ABB RobotStudio station: sesion2_parte1.rspag

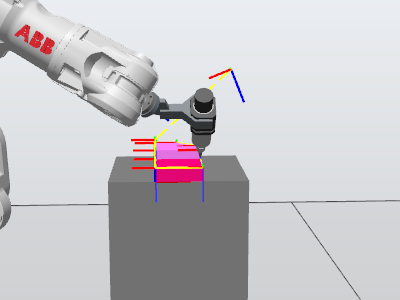
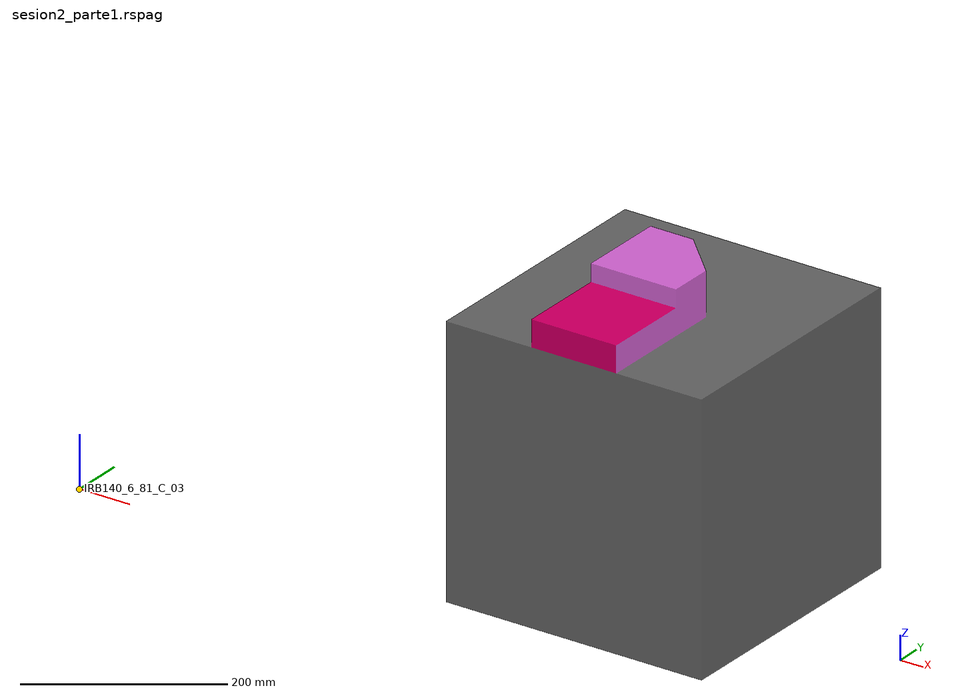
[picture v1: parts stored in the station drawn from their meshes, with robot base, taught points and paths (robot models come from the ABB library and are not in the file)]
--- station ---
Station sesion2 (saved by RobotStudio 24.1.10713.1)
Controller Controlador2
  mechanical unit ROB_1: IRB140_6_81_C_03, 6 joints, base frame (0, 0, 0) mm
Layout (positions relative to the parent item):
  - IRB140_6_81_C_03 [mechanism, from %ABB.RobotStudio.Models.IRB140%\IRB140_6_81_C_G_03.rslib] at (0, 0, 0) mm; joint values [-0.1632, 0.2338, 0.3026, 1.2516, 0.7538, -0.7373] (rad or m)
  - MyTool [mechanism, from Training Objects\myTool.rslib] at (513.67, -41.8, 471.8) mm, rotated rx 128.24 ry 25.81 rz 151.08 deg
  - Pieza_1 [part], size 300 x 300 x 300 mm
  - Pieza_7 [part], size 100 x 200 x 50 mm
Attachment: MyTool is attached to IRB140_6_81_C_03 / Link6
Attachment: Workobject_1 is attached to Pieza_7
Targets, tools, work objects and paths stored in the station and not in the controller backup, written as RAPID:
! task T_ROB1
MODULE CalibData
  PERS tooldata MyTool:=[TRUE,[[31.792631019,0,229.638935148],[0.945518576,0,0.325568154,0]],[1,[0,0,1],[1,0,0,0],0,0,0]];
  TASK PERS wobjdata Workobject_1:=[FALSE,TRUE,"",[[530,0,300],[1,0,0,0]],[[0,0,0],[1,0,0,0]]];
ENDMODULE

! task T_ROB1
MODULE Module1
  CONST robtarget Target_10:=[[0,0,30],[0,0,1,0],[0,0,-1,0],[9E+09,9E+09,9E+09,9E+09,9E+09,9E+09]];
  CONST robtarget Target_20:=[[100,0,30],[0,0,1,0],[0,0,-1,0],[9E+09,9E+09,9E+09,9E+09,9E+09,9E+09]];
  CONST robtarget Target_30:=[[100,100,30],[0,0,1,0],[0,-1,0,0],[9E+09,9E+09,9E+09,9E+09,9E+09,9E+09]];
  CONST robtarget Target_40:=[[100,100,50],[0,0,1,0],[0,-1,0,0],[9E+09,9E+09,9E+09,9E+09,9E+09,9E+09]];
  CONST robtarget Target_50:=[[100,150,50],[0,0,1,0],[0,-1,0,0],[9E+09,9E+09,9E+09,9E+09,9E+09,9E+09]];
  CONST robtarget Target_60:=[[50,200,50],[0,0,1,0],[0,-1,0,0],[9E+09,9E+09,9E+09,9E+09,9E+09,9E+09]];
  CONST robtarget Target_70:=[[0,200,50],[0,0,1,0],[0,-1,0,0],[9E+09,9E+09,9E+09,9E+09,9E+09,9E+09]];
  CONST robtarget Target_80:=[[0,100,50],[0,0,1,0],[0,-1,0,0],[9E+09,9E+09,9E+09,9E+09,9E+09,9E+09]];
  CONST robtarget Target_90:=[[0,100,30],[0,0,1,0],[0,-1,0,0],[9E+09,9E+09,9E+09,9E+09,9E+09,9E+09]];
  CONST robtarget pAprox:=[[0,0,90],[0,0,1,0],[0,0,-1,0],[9E+09,9E+09,9E+09,9E+09,9E+09,9E+09]];
  CONST robtarget pReposo:=[[689.268566117,0,537.147256028],[0.190808934,0,0.981627195,0],[0,0,0,0],[9E+09,9E+09,9E+09,9E+09,9E+09,9E+09]];
  CONST robtarget Target_30_Girado:=[[100,100,30],[0,0,0.923879533,0.382683432],[-1,0,-1,0],[9E+09,9E+09,9E+09,9E+09,9E+09,9E+09]];
  CONST robtarget Target_40_girado:=[[100,100,50],[0,0,0.923879533,0.382683432],[-1,0,-1,0],[9E+09,9E+09,9E+09,9E+09,9E+09,9E+09]];
  PROC Path_10()
    MoveJ pReposo,v1500,z100,MyTool\WObj:=wobj0;
    MoveJ pAprox,v1000,z100,MyTool\WObj:=Workobject_1;
    MoveL Target_10,v50,z0,MyTool\WObj:=Workobject_1;
    MoveL Target_20,v50,z0,MyTool\WObj:=Workobject_1;
    MoveL Target_30,v50,z0,MyTool\WObj:=Workobject_1;
    MoveL Target_30_Girado,v10,z0,MyTool\WObj:=Workobject_1;
    MoveL Target_40_girado,v50,z0,MyTool\WObj:=Workobject_1;
    MoveL Target_40,v50,z0,MyTool\WObj:=Workobject_1;
    MoveL Target_50,v50,z0,MyTool\WObj:=Workobject_1;
    MoveL Target_60,v50,z0,MyTool\WObj:=Workobject_1;
    MoveL Target_70,v50,z0,MyTool\WObj:=Workobject_1;
    MoveL Target_80,v50,z0,MyTool\WObj:=Workobject_1;
    MoveL Target_90,v50,z0,MyTool\WObj:=Workobject_1;
    MoveL Target_10,v50,z0,MyTool\WObj:=Workobject_1;
    MoveL pAprox,v50,z0,MyTool\WObj:=Workobject_1;
    MoveJ pReposo,v1000,z100,MyTool\WObj:=wobj0;
  ENDPROC
ENDMODULE


--- Backups/Controlador2/RAPID/TASK1/PROGMOD/Module1.mod ---
MODULE Module1
    !***********************************************************
    !
    ! M?dulo:  Module1
    !
    ! Descripción:
    !   <Introduzca la descripción aquí>
    !
    ! Autor: yisus
    !
    ! Versión: 1.0
    !
    !***********************************************************


    !***********************************************************
    !
    ! Procedimiento Main
    !
    !   Este es el punto de entrada de su programa
    !
    !***********************************************************
    PROC main()
        !Add your code here
    ENDPROC
ENDMODULE
